FUNCTION BOOL_TO_STRING_LHeaterON : STRING
VAR_INPUT
	nHeaterNumber	: INT;
	bON				: BOOL;
END_VAR
VAR
	sString			: STRING;
	sHeaterNumber	: STRING;
END_VAR

//LH: Line Heater x 8EA -> 8Channel TIC 1EA
//Model: HANYOUNG NUX, MC9-8RD0SS32

//STRING : '$0201DWR,02,0302(CH_NO),0001(CH_1),0501(AT),0001(AT-ON)
sString := '$0201DWR,02,0302,,0501,000$0D$0A';

//Convert to Channel from Heater Number
sHeaterNumber := DINT_TO_DECSTR(nHeaterNumber, 4);
sString := INSERT(sString,sHeaterNumber,15);

IF bON = TRUE THEN
	sString := INSERT(sString,'1',28);
ELSE
	sString := INSERT(sString,'0',28);
END_IF

BOOL_TO_STRING_LHeaterON := sString;

END_FUNCTION

(* stored: Version 1.1.0.1, ProductVersion 3.1.4024.12
   POU BOOL_TO_STRING_LHeaterON: Id {ab6dfe8d-8c1e-4695-a9b3-243912508813}, SpecialFunc None *)
